# EPICS autosave request: iocBoot/ioc13idd_micromax1/auto_settings.req
file "ccd_settings.req", P=13IDDMicroMax1:, C=det1:
